{attribute 'qualified_only'}
{attribute 'to_string'}
// Default CHAN 1, add 0x800 next channel
TYPE E_Module :
(
    CHAN1	:= 1,
    CHAN2	:= 2,
    CHAN3	:= 3
) WORD;
END_TYPE

(* stored: Version 1.1.0.1
   DUT E_Module: Id {2ec85200-d340-4d87-8d2a-acaf2cf7f4d9} *)
